// TIA Portal V17 export
// export: Created 2023-12-22T15:08:03.2766078Z, ExportSetting WithDefaults, DisplayName Totally Integrated Automation Portal, DisplayVersion V17, DisplayName TIA Portal Openness, DisplayVersion V17, DisplayName TIA Portal Version Control Interface, DisplayVersion V17, DisplayName STEP 7 Professional, DisplayVersion V17, DisplayName STEP 7 Safety, DisplayVersion V17, DisplayName WinCC Advanced, DisplayVersion V17
DATA_BLOCK "P_6_DB"   // DB605
VERSION : 0.1
// stored: AutoNumber false, DBAccessibleFromOPCUA true, DBAccessibleFromWebserver true, InstanceOfName DRV_M_DA, InstanceOfType FB
"DRV_M_DA"
   // VAR_INPUT
   //    All_Block : Bool;
   // END_VAR
   // VAR_IN_OUT
   //    FB_QF : Bool;
   //    FB_KM : Bool;
   //    S_Alarm : Bool;
   //    CMD_Run : Bool;
   // END_VAR
   // VAR RETAIN
   //    CMD : "CMD";
   //    Mode : Int;
   //    Status : Int;
   //    Use : Struct
   //       QF { S7_SetPoint := 'True'} : Bool := TRUE;
   //       KM { S7_SetPoint := 'True'} : Bool := TRUE;
   //       OpTime { S7_SetPoint := 'True'} : Bool := TRUE;
   //       Analog { S7_SetPoint := 'True'} : Bool := TRUE;
   //       Local_Keys : Bool;
   //    END_STRUCT;
   //    FB : Struct
   //       QF : Bool;
   //       KM : Bool;
   //       Local_Start : Bool;
   //       Local_Stop : Bool;
   //    END_STRUCT;
   //    ON : Bool;
   //    OFF : Bool;
   //    Tx { S7_SetPoint := 'True'} : Array[0..3] of "Time_S";
   //    Inv : Struct
   //       CMD { S7_SetPoint := 'True'} : Bool := FALSE;
   //       QF { S7_SetPoint := 'True'} : Bool := FALSE;
   //       KM { S7_SetPoint := 'True'} : Bool := FALSE;
   //    END_STRUCT;
   //    Alarm : Struct
   //       Block : Bool;
   //       QF : Bool;
   //       Start : Bool;
   //       Stop : Bool;
   //       Termo : Bool;
   //       Alarm : Bool;
   //       Safety : Bool;
   //       OpTime : Bool;
   //       C_Max : Bool;
   //       C_Error : Bool;
   //    END_STRUCT;
   //    Alarms : Word;
   //    Events : Word;
   //    pos : Array[0..15] of Bool;
   //    OpTime_h : DInt;
   //    OpTime_s { S7_SetPoint := 'True'} : DInt := 4026605;
   //    OpTime_SP { S7_SetPoint := 'True'} : DInt := 2160;
   //    OpTime_Now_h : DInt;
   //    OpTime_Now_s { S7_SetPoint := 'True'} : DInt := 4026605;
   //    CodeID { S7_SetPoint := 'True'} : Int := 0;
   //    Indirect : Struct
   //       FB_QF { S7_SetPoint := 'True'} : Bool := TRUE;
   //       FB_KM { S7_SetPoint := 'True'} : Bool := TRUE;
   //       CMD { S7_SetPoint := 'True'} : Bool := TRUE;
   //    END_STRUCT;
   //    Indirect_BYTE : Struct
   //       FB_QF { S7_SetPoint := 'True'} : Int := 1;
   //       FB_KM { S7_SetPoint := 'True'} : Int := 1;
   //       CMD { S7_SetPoint := 'True'} : Int := 0;
   //    END_STRUCT;
   //    Indirect_BIT : Struct
   //       FB_QF { S7_SetPoint := 'True'} : Int := 2;
   //       FB_KM { S7_SetPoint := 'True'} : Int := 3;
   //       CMD { S7_SetPoint := 'True'} : Int := 5;
   //    END_STRUCT;
   //    SP_A : Real;
   //    SP_M : Real;
   //    ADDR { S7_SetPoint := 'True'} : Int := 266;
   //    Converter { S7_SetPoint := 'True'} : "Converter_LAD";
   //    VmA : Real;
   //    Output_Type { S7_SetPoint := 'True'} : Int := 0;
   //    "Type" { S7_SetPoint := 'True'} : Int := 1;
   //    Slow { S7_SetPoint := 'True'} : "Slow";
   //    C : Real;
   //    C_Max { S7_SetPoint := 'True'} : Real := 0.0;
   //    T_С { S7_SetPoint := 'True'} : "Time_S";
   //    Time_DTL { S7_SetPoint := 'True'} : DTL := DTL#2023-02-16-09:35:05.181284915;
   // END_VAR
BEGIN
   Tx[0..1].SP := 0;
   Tx[2].SP := 2;
   Tx[3].SP := 90;
   Converter.Use_Min_In := FALSE;
   Converter.Use_Max_In := FALSE;
   Converter.Use_Min_Out := FALSE;
   Converter.Use_Max_Out := FALSE;
   Converter.IO := FALSE;
   Converter.Inverse := FALSE;
   Converter.Min_In := 0.0;
   Converter.Min_Out := 0.0;
   Converter.Max_In := 50.0;
   Converter.Max_Out := 27645.0;
   Slow.Use_Up := TRUE;
   Slow.Use_Down := TRUE;
   Slow.Step_Up := 0.005;
   Slow.Step_Down := 0.05;
   Slow.T_Up.SP := 0.1;
   Slow.T_Up.One := 0.1;
   Slow.T_Down.SP := 0.1;
   Slow.T_Down.One := 0.1;
   T_С.SP := 2;
END_DATA_BLOCK
